FUNCTION_BLOCK REAL_Param
VAR_INPUT PERSISTENT
	val			: REAL;
END_VAR

END_FUNCTION_BLOCK

(* stored: Version 1.1.0.1
   POU REAL_Param: Id {f3423309-7861-4f43-9521-886eabbb168d}, SpecialFunc None *)
